// TIA Portal V20 export
FUNCTION "PostProcessing" : Void   // FC57, LAD
TITLE = Post Processing
// V1.0  25.05.04  Safety test program: sending data via F-link
// stored: Namespace Safety, SetENOAutomatically false
BEGIN

REGION Network 1: Sending data to BA030, stacker #1
   // V1.0  25.05.04  Safety test program: FlinkSendToBA30AC1
   //                 Send ID: 102, Receive ID: 103
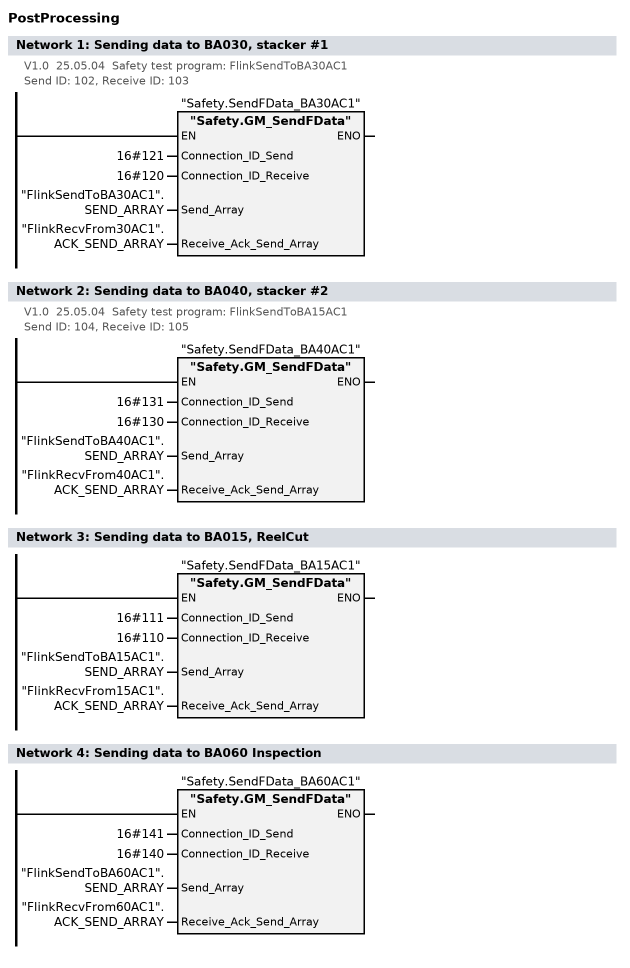
   RUNG wire#powerrail
      "Safety.SendFData_BA30AC1"(Connection_ID_Send := 16#121, Connection_ID_Receive := 16#120, Send_Array := "FlinkSendToBA30AC1".SEND_ARRAY, Receive_Ack_Send_Array := "FlinkRecvFrom30AC1".ACK_SEND_ARRAY)
   END_RUNG
   // the same network as SCL:
   "Safety.SendFData_BA30AC1"(Connection_ID_Send := 16#121,   // "Safety.GM_SendFData"
                           Connection_ID_Receive := 16#120,
                           Send_Array := "FlinkSendToBA30AC1".SEND_ARRAY,
                           Receive_Ack_Send_Array := "FlinkRecvFrom30AC1".ACK_SEND_ARRAY);
END_REGION

REGION Network 2: Sending data to BA040, stacker #2
   // V1.0  25.05.04  Safety test program: FlinkSendToBA15AC1
   //                 Send ID: 104, Receive ID: 105
   RUNG wire#powerrail
      "Safety.SendFData_BA40AC1"(Connection_ID_Send := 16#131, Connection_ID_Receive := 16#130, Send_Array := "FlinkSendToBA40AC1".SEND_ARRAY, Receive_Ack_Send_Array := "FlinkRecvFrom40AC1".ACK_SEND_ARRAY)
   END_RUNG
   // the same network as SCL:
   "Safety.SendFData_BA40AC1"(Connection_ID_Send := 16#131,   // "Safety.GM_SendFData"
                           Connection_ID_Receive := 16#130,
                           Send_Array := "FlinkSendToBA40AC1".SEND_ARRAY,
                           Receive_Ack_Send_Array := "FlinkRecvFrom40AC1".ACK_SEND_ARRAY);
END_REGION

REGION Network 3: Sending data to BA015, ReelCut
   RUNG wire#powerrail
      "Safety.SendFData_BA15AC1"(Connection_ID_Send := 16#111, Connection_ID_Receive := 16#110, Send_Array := "FlinkSendToBA15AC1".SEND_ARRAY, Receive_Ack_Send_Array := "FlinkRecvFrom15AC1".ACK_SEND_ARRAY)
   END_RUNG
   // the same network as SCL:
   "Safety.SendFData_BA15AC1"(Connection_ID_Send := 16#111,   // "Safety.GM_SendFData"
                           Connection_ID_Receive := 16#110,
                           Send_Array := "FlinkSendToBA15AC1".SEND_ARRAY,
                           Receive_Ack_Send_Array := "FlinkRecvFrom15AC1".ACK_SEND_ARRAY);
END_REGION

REGION Network 4: Sending data to BA060 Inspection
   RUNG wire#powerrail
      "Safety.SendFData_BA60AC1"(Connection_ID_Send := 16#141, Connection_ID_Receive := 16#140, Send_Array := "FlinkSendToBA60AC1".SEND_ARRAY, Receive_Ack_Send_Array := "FlinkRecvFrom60AC1".ACK_SEND_ARRAY)
   END_RUNG
   // the same network as SCL:
   "Safety.SendFData_BA60AC1"(Connection_ID_Send := 16#141,   // "Safety.GM_SendFData"
                           Connection_ID_Receive := 16#140,
                           Send_Array := "FlinkSendToBA60AC1".SEND_ARRAY,
                           Receive_Ack_Send_Array := "FlinkRecvFrom60AC1".ACK_SEND_ARRAY);
END_REGION

REGION Network 5 (SCL)
   "Safety.DataToSafety".ackSafetyFromHmi := "Safety.DataFromStandard".ackSafetyFromHmi;
   "Safety.DataFromSafety".ackOP_changeRequired := "Safety.InstMain_Safety_RTG1".instAckOP.Q;
END_REGION
END_FUNCTION
